// TIA Portal project "TIA portal v16_V16" (V16)
// Vorlageprojekt für das Buch mit Zielsystem S7-1200

(* hardware
DEVICE "S7-1200 station_1"  S7-1200 Station
   slot 0: "Rack_0"  S7-1200 Rack  Rack  V1.0
   slot 1: "PLC_2"  CPU 1215C DC/DC/DC  6ES7 215-1AG40-0XB0  V4.4
   slot 2: "DI 16/DQ 16x24VDC_1"  6ES7 223-1BL32-0XB0  V2.0
   slot 3: "DI 16x24VDC_1"  6ES7 221-1BH32-0XB0  V2.0
   slot 4: "AI 4x13BIT/AQ 2x14BIT_1"  6ES7 234-4HE32-0XB0  V2.1
*)

// ===== PLC "PLC_2"  CPU 1215C DC/DC/DC =====

VAR_GLOBAL   // PLC tag table "Default tag table"
   "Security Relay" AT %I0.0 : Bool;
   "Emergency stop feeding" AT %I0.1 : Bool;
   "Emergency stop elevator" AT %I0.2 : Bool;
   "Emergency stop load beld" AT %I0.3 : Bool;
   "Select auto" AT %I0.4 : Bool;
   "Select manual" AT %I0.5 : Bool;
   "Fault reset button" AT %I0.6 : Bool;
   "Manual box feeding button" AT %I1.0 : Bool;
   "Manual load beld" AT %I1.1 : Bool;
   "Manual Clamp" AT %I1.2 : Bool;
   "Box feeder motor guard" AT %I2.0 : Bool;
   "Enable load beld motor guard" AT %I2.1 : Bool;
   "Elevator motor guard" AT %I2.2 : Bool;
   "Load pallet motor guard" AT %I2.3 : Bool;
   "Pallet feeder motor guard" AT %I2.4 : Bool;
   "Exit conveyor motor guard" AT %I2.5 : Bool;
   "Box feeder motor feedback" AT %I3.0 : Bool;
   "Enable load beld motor feedback" AT %I3.1 : Bool;
   "Elevator motor feedback up" AT %I3.2 : Bool;
   "Elevator motor feedback down" AT %I3.3 : Bool;
   "Load pallet motor feedback" AT %I3.4 : Bool;
   "Pallet feeder motor feedback" AT %I3.5 : Bool;
   "Exit conveyor motor feedback" AT %I3.6 : Bool;
   "Pallet at entry" AT %I4.0 : Bool;
   "Pallet at exit" AT %I4.1 : Bool;
   "Pallet loaded" AT %I4.2 : Bool;
   "Up load pallet" AT %I4.3 : Bool;
   "Down load pallet" AT %I4.4 : Bool;
   "Box at entry" AT %I4.5 : Bool;
   "Pusher limit" AT %I4.6 : Bool;
   "Plate limit" AT %I4.7 : Bool;
   "Clamped" AT %I5.0 : Bool;
   "Relay warning ligth" AT %Q0.0 : Bool;
   "Relay aux turn valve" AT %Q0.1 : Bool;
   "Relay aux push valve" AT %Q0.2 : Bool;
   "Relay aux plate valve" AT %Q0.3 : Bool;
   "Relay Clamp" AT %Q0.4 : Bool;
   "Move to limit" AT %Q0.5 : Bool;
   "Enable pallet emiter" AT %Q0.6 : Bool;
   "Enable exit conveyor" AT %Q0.7 : Bool;
   "Enable box feeder motor" AT %Q2.0 : Bool;
   "Enable load beld motor" AT %Q2.1 : Bool;
   "Enable elevator up motor" AT %Q2.2 : Bool;
   "Enable elevator down motor" AT %Q2.3 : Bool;
   "Enable Load pallet motor" AT %Q2.4 : Bool;
   "Enable Pallet feeder motor" AT %Q2.5 : Bool;
   "Enable exit conveyor motor" AT %Q2.6 : Bool;
   "Fault reset light" AT %Q3.0 : Bool;
   "Start feeding light" AT %Q3.1 : Bool;
   "Stop feeding light" AT %Q3.2 : Bool;
   "Counter box" AT %QW50 : Word;
   "Input_Security_Relay" AT %M0.0 : Bool;
   "Input_Emergency_stop_feeding" AT %M0.1 : Bool;
   "Input_emergency_stop_elevator" AT %M0.2 : Bool;
   "Input_emergency_stop_load_beld" AT %M0.3 : Bool;
   "Input_select_auto" AT %M0.4 : Bool;
   "Input_select_manual" AT %M0.5 : Bool;
   "Input_Fault_reset_button" AT %M0.6 : Bool;
   "Input_manual_box_feeding_button" AT %M1.0 : Bool;
   "Input_manual_load_beld" AT %M1.1 : Bool;
   "Input_manual_clamp" AT %M1.2 : Bool;
   "Input_manual_pallet_feeder" AT %M1.3 : Bool;
   "Input_box_feeder_motor_guard" AT %M2.0 : Bool;
   "Input_enable_load_beld_motor_guard" AT %M2.1 : Bool;
   "Input_elevator_motor_guard" AT %M2.2 : Bool;
   "Input_load_pallet_motor_guard" AT %M2.3 : Bool;
   "Input_pallet_feeder_motor_guad" AT %M2.4 : Bool;
   "Input_box_feeder_motor_feedback" AT %M3.0 : Bool;
   "Input_enable_load_beld_motor_feedback" AT %M3.1 : Bool;
   "Input_elevator_motor_feedback_up" AT %M3.2 : Bool;
   "Input_elevator_motor_feedback_down" AT %M3.3 : Bool;
   "Input_load_pallet_motor_feedback" AT %M3.4 : Bool;
   "Input_pallet_feeder_motor_feedback" AT %M3.5 : Bool;
   "Input_pallet_at_entry" AT %M4.0 : Bool;
   "Input_pallet_at_exit" AT %M4.1 : Bool;
   "Input_pallet_loaded" AT %M4.2 : Bool;
   "Input_up_load_pallet" AT %M4.3 : Bool;
   "Input_down_load_pallet" AT %M4.4 : Bool;
   "Input_box_at_entry" AT %M4.5 : Bool;
   "Input_pusher_limit" AT %M4.6 : Bool;
   "Input_plate_limit" AT %M4.7 : Bool;
   "Input_clamped" AT %M5.0 : Bool;
   "Output_warning_ligth" AT %M10.0 : Bool;
   "Output_relay_aux_turn_valve" AT %M10.1 : Bool;
   "Ouput_relay_aux_push_valve" AT %M10.2 : Bool;
   "Output_relay_aux_plate_valve" AT %M10.3 : Bool;
   "Output_relay_clamp" AT %M10.4 : Bool;
   "Ouput_move_to_limit" AT %M10.5 : Bool;
   "Output_enable_pallet_emiter" AT %M10.6 : Bool;
   "Output_enable_exit_conveyor" AT %M10.7 : Bool;
   "Output_enable_box_feeder_motor" AT %M12.0 : Bool;
   "Output_enable_load_beld_motor" AT %M12.1 : Bool;
   "Output_enable_elevator_up_motor" AT %M12.2 : Bool;
   "Output_enable_elevator_down_motor" AT %M12.3 : Bool;
   "Output_enable_load_pallet_motor" AT %M12.4 : Bool;
   "Output_enable_pallet_feeder_motor" AT %M12.5 : Bool;
   "Output_enable_exit_conveyor_motor" AT %M12.6 : Bool;
   "Output_fault_reset_light" AT %M13.0 : Bool;
   "Output_start_feeding_light" AT %M13.1 : Bool;
   "Output_stop_feeding_light" AT %M13.2 : Bool;
   "Ouput_counter_box" AT %MW100 : Word;
   "Emergency_enable" AT %M30.0 : Bool;
   "Manual_box_feeding_drive" AT %M30.1 : Bool;
   "Manual pallet feeder" AT %I1.3 : Bool;
   "Manual load pallet" AT %I1.4 : Bool;
   "Input_manual_load_pallet" AT %M1.4 : Bool;
   "Input_manual_exit_conveyor" AT %M1.5 : Bool;
   "Manual_load_beld_drive" AT %M30.2 : Bool;
   "Manual_clamp_drive" AT %M30.3 : Bool;
   "Manual_pallet_feeder_drive" AT %M30.4 : Bool;
   "Elevator moving" AT %I5.1 : Bool;
   "Manual exit conveyor" AT %I1.5 : Bool;
   "Manual elevator up" AT %I5.2 : Bool;
   "Manual elevator down" AT %I5.3 : Bool;
   "Input_elevator_moving" AT %M5.1 : Bool;
   "Input_manual_elevator_up" AT %M5.2 : Bool;
   "Input_manual_elevator_down" AT %M5.3 : Bool;
   "Manual_load_pallet_drive" AT %M30.5 : Bool;
   "Manual_exit_conveyor_drive" AT %M30.6 : Bool;
   "Manual_elevator_up_drive" AT %M30.7 : Bool;
   "Manual_elevator_down_drive" AT %M31.0 : Bool;
   "Input_exit_conveyor_motor_guard" AT %M2.5 : Bool;
   "Input_exit_conveyor_motor_feedback" AT %M3.6 : Bool;
   "Aux_manual_box_feeding_drive" AT %M31.1 : Bool;
   "Up_manual_box_feeding_drive" AT %M6.0 : Bool;
   "Up_manual_load_beld_drive" AT %M6.1 : Bool;
   "Aux_manual_load_beld_drive" AT %M31.2 : Bool;
   "Aux_manual_pallet_feeder_drive" AT %M31.4 : Bool;
   "Aux_manual_load_pallet_drive" AT %M31.5 : Bool;
   "Aux_manual_exit_conveyor_drive" AT %M31.6 : Bool;
   "Aux_manual_elevator_up_drive" AT %M31.7 : Bool;
   "Aux_manual_elevator_down_drive" AT %M32.0 : Bool;
   "Up_manual_pallet_feeder_drive" AT %M6.2 : Bool;
   "Up_manual_load_pallet_drive" AT %M6.3 : Bool;
   "Up_manual_exit_conveyor_drive" AT %M6.4 : Bool;
   "Up_manual_elevator_up_drive" AT %M6.5 : Bool;
   "Up_manual_elevator_down_drive" AT %M6.6 : Bool;
END_VAR

DATA_BLOCK "Engine_starter_DB_box_feeder"   // DB1
{ S7_Optimized_Access := 'TRUE' }
VERSION : 0.1
// stored: InstanceOfName Engine_starter
"Engine_starter"
BEGIN
END_DATA_BLOCK

DATA_BLOCK "Engine_starter_DB_load_beld"   // DB2
{ S7_Optimized_Access := 'TRUE' }
VERSION : 0.1
// stored: InstanceOfName Engine_starter
"Engine_starter"
BEGIN
END_DATA_BLOCK

DATA_BLOCK "Engine_starter_DB_elevator_up"   // DB3
{ S7_Optimized_Access := 'TRUE' }
VERSION : 0.1
// stored: InstanceOfName Engine_starter
"Engine_starter"
BEGIN
END_DATA_BLOCK

DATA_BLOCK "Engine_starter_DB_elevator_down"   // DB4
{ S7_Optimized_Access := 'TRUE' }
VERSION : 0.1
// stored: InstanceOfName Engine_starter
"Engine_starter"
BEGIN
END_DATA_BLOCK

DATA_BLOCK "Engine_starter_DB_load_pallet"   // DB5
{ S7_Optimized_Access := 'TRUE' }
VERSION : 0.1
// stored: InstanceOfName Engine_starter
"Engine_starter"
BEGIN
END_DATA_BLOCK

DATA_BLOCK "Engine_starter_DB_pallet_feeder"   // DB6
{ S7_Optimized_Access := 'TRUE' }
VERSION : 0.1
// stored: InstanceOfName Engine_starter
"Engine_starter"
BEGIN
END_DATA_BLOCK

DATA_BLOCK "Engine_starter_DB_exit_conveyor"   // DB7
{ S7_Optimized_Access := 'TRUE' }
VERSION : 0.1
// stored: InstanceOfName Engine_starter
"Engine_starter"
BEGIN
END_DATA_BLOCK

FUNCTION_BLOCK "Engine_starter"   // FB1, LAD
{ S7_Optimized_Access := 'TRUE' }
VERSION : 0.1
   VAR_INPUT
      STOP_EMERGENCY : Bool;
      THERMAL_SHUTDOWN : Bool;
      CONTACT_FEEDBACK : Bool;
      ENABLE : Bool;
      RESET_FAULT : Bool;
   END_VAR
   VAR_OUTPUT
      START_ENABLED : Bool;
      STARTING_FAILURE : Bool;
      ACTIVE_EMERGENCY : Bool;
      ACTIVE_THERMAL : Bool;
      FEEDBACK_FAILURE : Bool;
   END_VAR
   VAR
      stop_error : Bool;
      temp_feedback : TON_TIME;
      enable_engine : Bool;
      temp_thermal_shutdown : TON_TIME;
   END_VAR
BEGIN

REGION Network 1
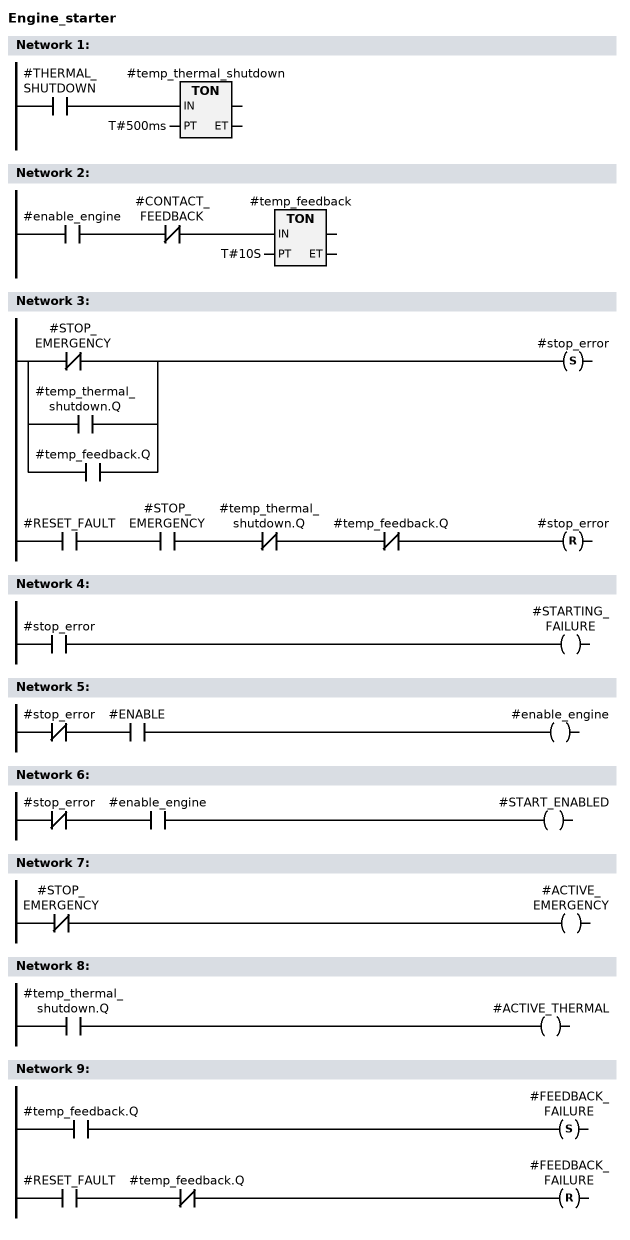
   #temp_thermal_shutdown(IN := #THERMAL_SHUTDOWN, PT := T#500ms);   // TON
END_REGION

REGION Network 2
   #temp_feedback(IN := #enable_engine AND NOT #CONTACT_FEEDBACK, PT := T#10S);   // TON
END_REGION

REGION Network 3
   RUNG wire#powerrail
      I_Contact( #STOP_EMERGENCY )
      wire#w1
      S_Coil( #stop_error )
   END_RUNG
   RUNG wire#powerrail
      Contact( #temp_thermal_shutdown.Q )
   END_RUNG wire#w1
   RUNG wire#powerrail
      Contact( #temp_feedback.Q )
   END_RUNG wire#w1
   RUNG wire#powerrail
      Contact( #RESET_FAULT )
      Contact( #STOP_EMERGENCY )
      I_Contact( #temp_thermal_shutdown.Q )
      I_Contact( #temp_feedback.Q )
      R_Coil( #stop_error )
   END_RUNG
   // the same network as SCL:
   IF NOT #STOP_EMERGENCY OR #temp_thermal_shutdown.Q OR #temp_feedback.Q THEN #stop_error := TRUE; END_IF;
   IF #RESET_FAULT AND #STOP_EMERGENCY AND NOT #temp_thermal_shutdown.Q AND NOT #temp_feedback.Q THEN
       #stop_error := FALSE;
   END_IF;
END_REGION

REGION Network 4
   RUNG wire#powerrail
      Contact( #stop_error )
      Coil( #STARTING_FAILURE )
   END_RUNG
   // the same network as SCL:
   #STARTING_FAILURE := #stop_error;
END_REGION

REGION Network 5
   RUNG wire#powerrail
      I_Contact( #stop_error )
      Contact( #ENABLE )
      Coil( #enable_engine )
   END_RUNG
   // the same network as SCL:
   #enable_engine := NOT #stop_error AND #ENABLE;
END_REGION

REGION Network 6
   RUNG wire#powerrail
      I_Contact( #stop_error )
      Contact( #enable_engine )
      Coil( #START_ENABLED )
   END_RUNG
   // the same network as SCL:
   #START_ENABLED := NOT #stop_error AND #enable_engine;
END_REGION

REGION Network 7
   RUNG wire#powerrail
      I_Contact( #STOP_EMERGENCY )
      Coil( #ACTIVE_EMERGENCY )
   END_RUNG
   // the same network as SCL:
   #ACTIVE_EMERGENCY := NOT #STOP_EMERGENCY;
END_REGION

REGION Network 8
   RUNG wire#powerrail
      Contact( #temp_thermal_shutdown.Q )
      Coil( #ACTIVE_THERMAL )
   END_RUNG
   // the same network as SCL:
   #ACTIVE_THERMAL := #temp_thermal_shutdown.Q;
END_REGION

REGION Network 9
   RUNG wire#powerrail
      Contact( #temp_feedback.Q )
      S_Coil( #FEEDBACK_FAILURE )
   END_RUNG
   RUNG wire#powerrail
      Contact( #RESET_FAULT )
      I_Contact( #temp_feedback.Q )
      R_Coil( #FEEDBACK_FAILURE )
   END_RUNG
   // the same network as SCL:
   IF #temp_feedback.Q THEN #FEEDBACK_FAILURE := TRUE; END_IF;
   IF #RESET_FAULT AND NOT #temp_feedback.Q THEN #FEEDBACK_FAILURE := FALSE; END_IF;
END_REGION
END_FUNCTION_BLOCK

FUNCTION "Input_Management" : Void   // FC1, LAD
{ S7_Optimized_Access := 'TRUE' }
VERSION : 0.1
BEGIN

REGION Network 1
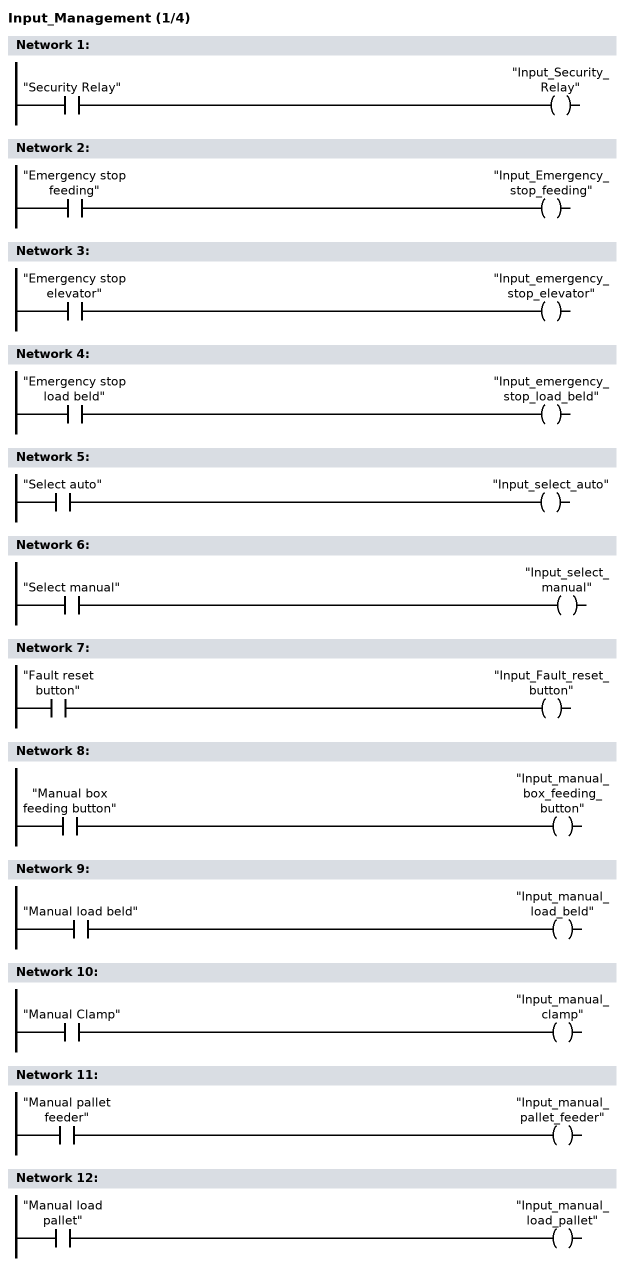
   RUNG wire#powerrail
      Contact( "Security Relay" )
      Coil( "Input_Security_Relay" )
   END_RUNG
   // the same network as SCL:
   "Input_Security_Relay" := "Security Relay";
END_REGION

REGION Network 2
   RUNG wire#powerrail
      Contact( "Emergency stop feeding" )
      Coil( "Input_Emergency_stop_feeding" )
   END_RUNG
   // the same network as SCL:
   "Input_Emergency_stop_feeding" := "Emergency stop feeding";
END_REGION

REGION Network 3
   RUNG wire#powerrail
      Contact( "Emergency stop elevator" )
      Coil( "Input_emergency_stop_elevator" )
   END_RUNG
   // the same network as SCL:
   "Input_emergency_stop_elevator" := "Emergency stop elevator";
END_REGION

REGION Network 4
   RUNG wire#powerrail
      Contact( "Emergency stop load beld" )
      Coil( "Input_emergency_stop_load_beld" )
   END_RUNG
   // the same network as SCL:
   "Input_emergency_stop_load_beld" := "Emergency stop load beld";
END_REGION

REGION Network 5
   RUNG wire#powerrail
      Contact( "Select auto" )
      Coil( "Input_select_auto" )
   END_RUNG
   // the same network as SCL:
   "Input_select_auto" := "Select auto";
END_REGION

REGION Network 6
   RUNG wire#powerrail
      Contact( "Select manual" )
      Coil( "Input_select_manual" )
   END_RUNG
   // the same network as SCL:
   "Input_select_manual" := "Select manual";
END_REGION

REGION Network 7
   RUNG wire#powerrail
      Contact( "Fault reset button" )
      Coil( "Input_Fault_reset_button" )
   END_RUNG
   // the same network as SCL:
   "Input_Fault_reset_button" := "Fault reset button";
END_REGION

REGION Network 8
   RUNG wire#powerrail
      Contact( "Manual box feeding button" )
      Coil( "Input_manual_box_feeding_button" )
   END_RUNG
   // the same network as SCL:
   "Input_manual_box_feeding_button" := "Manual box feeding button";
END_REGION

REGION Network 9
   RUNG wire#powerrail
      Contact( "Manual load beld" )
      Coil( "Input_manual_load_beld" )
   END_RUNG
   // the same network as SCL:
   "Input_manual_load_beld" := "Manual load beld";
END_REGION

REGION Network 10
   RUNG wire#powerrail
      Contact( "Manual Clamp" )
      Coil( "Input_manual_clamp" )
   END_RUNG
   // the same network as SCL:
   "Input_manual_clamp" := "Manual Clamp";
END_REGION

REGION Network 11
   RUNG wire#powerrail
      Contact( "Manual pallet feeder" )
      Coil( "Input_manual_pallet_feeder" )
   END_RUNG
   // the same network as SCL:
   "Input_manual_pallet_feeder" := "Manual pallet feeder";
END_REGION

REGION Network 12
   RUNG wire#powerrail
      Contact( "Manual load pallet" )
      Coil( "Input_manual_load_pallet" )
   END_RUNG
   // the same network as SCL:
   "Input_manual_load_pallet" := "Manual load pallet";
END_REGION

REGION Network 13
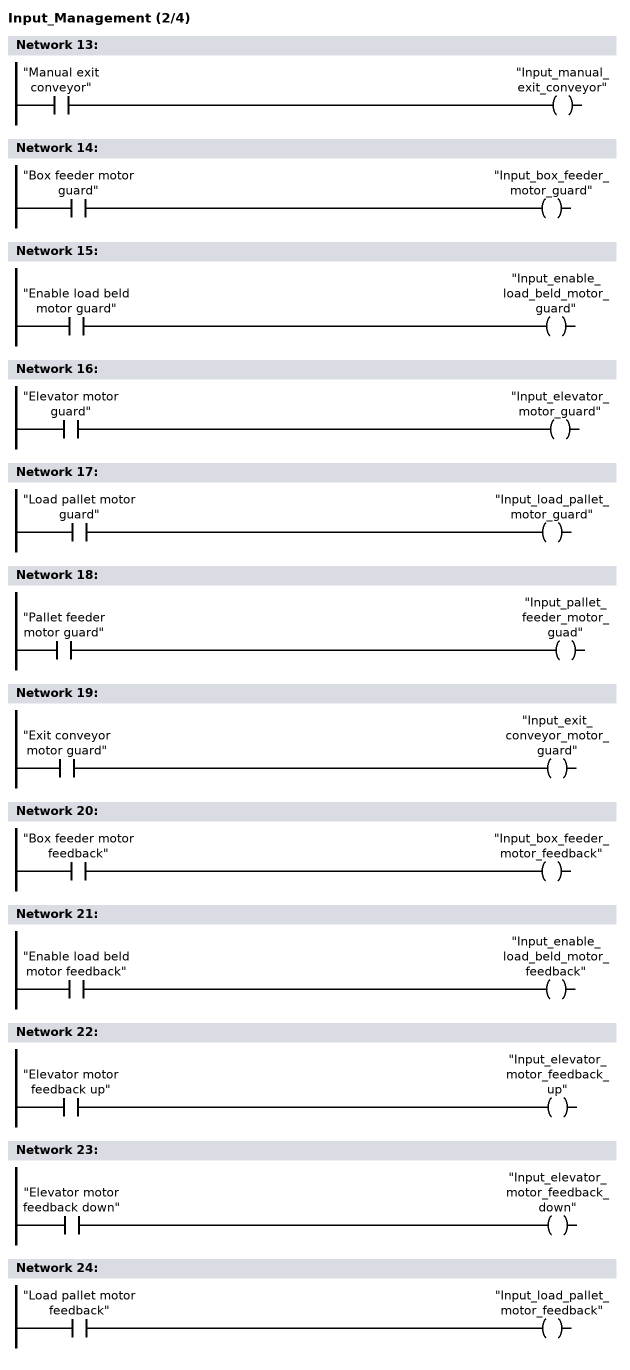
   RUNG wire#powerrail
      Contact( "Manual exit conveyor" )
      Coil( "Input_manual_exit_conveyor" )
   END_RUNG
   // the same network as SCL:
   "Input_manual_exit_conveyor" := "Manual exit conveyor";
END_REGION

REGION Network 14
   RUNG wire#powerrail
      Contact( "Box feeder motor guard" )
      Coil( "Input_box_feeder_motor_guard" )
   END_RUNG
   // the same network as SCL:
   "Input_box_feeder_motor_guard" := "Box feeder motor guard";
END_REGION

REGION Network 15
   RUNG wire#powerrail
      Contact( "Enable load beld motor guard" )
      Coil( "Input_enable_load_beld_motor_guard" )
   END_RUNG
   // the same network as SCL:
   "Input_enable_load_beld_motor_guard" := "Enable load beld motor guard";
END_REGION

REGION Network 16
   RUNG wire#powerrail
      Contact( "Elevator motor guard" )
      Coil( "Input_elevator_motor_guard" )
   END_RUNG
   // the same network as SCL:
   "Input_elevator_motor_guard" := "Elevator motor guard";
END_REGION

REGION Network 17
   RUNG wire#powerrail
      Contact( "Load pallet motor guard" )
      Coil( "Input_load_pallet_motor_guard" )
   END_RUNG
   // the same network as SCL:
   "Input_load_pallet_motor_guard" := "Load pallet motor guard";
END_REGION

REGION Network 18
   RUNG wire#powerrail
      Contact( "Pallet feeder motor guard" )
      Coil( "Input_pallet_feeder_motor_guad" )
   END_RUNG
   // the same network as SCL:
   "Input_pallet_feeder_motor_guad" := "Pallet feeder motor guard";
END_REGION

REGION Network 19
   RUNG wire#powerrail
      Contact( "Exit conveyor motor guard" )
      Coil( "Input_exit_conveyor_motor_guard" )
   END_RUNG
   // the same network as SCL:
   "Input_exit_conveyor_motor_guard" := "Exit conveyor motor guard";
END_REGION

REGION Network 20
   RUNG wire#powerrail
      Contact( "Box feeder motor feedback" )
      Coil( "Input_box_feeder_motor_feedback" )
   END_RUNG
   // the same network as SCL:
   "Input_box_feeder_motor_feedback" := "Box feeder motor feedback";
END_REGION

REGION Network 21
   RUNG wire#powerrail
      Contact( "Enable load beld motor feedback" )
      Coil( "Input_enable_load_beld_motor_feedback" )
   END_RUNG
   // the same network as SCL:
   "Input_enable_load_beld_motor_feedback" := "Enable load beld motor feedback";
END_REGION

REGION Network 22
   RUNG wire#powerrail
      Contact( "Elevator motor feedback up" )
      Coil( "Input_elevator_motor_feedback_up" )
   END_RUNG
   // the same network as SCL:
   "Input_elevator_motor_feedback_up" := "Elevator motor feedback up";
END_REGION

REGION Network 23
   RUNG wire#powerrail
      Contact( "Elevator motor feedback down" )
      Coil( "Input_elevator_motor_feedback_down" )
   END_RUNG
   // the same network as SCL:
   "Input_elevator_motor_feedback_down" := "Elevator motor feedback down";
END_REGION

REGION Network 24
   RUNG wire#powerrail
      Contact( "Load pallet motor feedback" )
      Coil( "Input_load_pallet_motor_feedback" )
   END_RUNG
   // the same network as SCL:
   "Input_load_pallet_motor_feedback" := "Load pallet motor feedback";
END_REGION

REGION Network 25
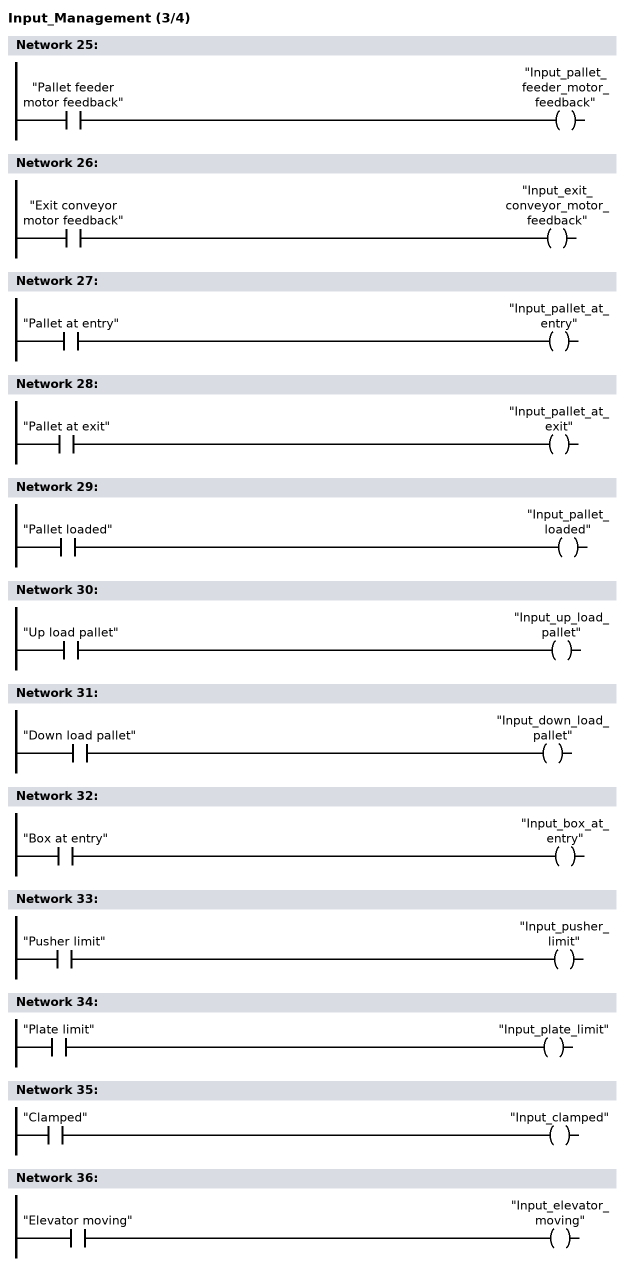
   RUNG wire#powerrail
      Contact( "Pallet feeder motor feedback" )
      Coil( "Input_pallet_feeder_motor_feedback" )
   END_RUNG
   // the same network as SCL:
   "Input_pallet_feeder_motor_feedback" := "Pallet feeder motor feedback";
END_REGION

REGION Network 26
   RUNG wire#powerrail
      Contact( "Exit conveyor motor feedback" )
      Coil( "Input_exit_conveyor_motor_feedback" )
   END_RUNG
   // the same network as SCL:
   "Input_exit_conveyor_motor_feedback" := "Exit conveyor motor feedback";
END_REGION

REGION Network 27
   RUNG wire#powerrail
      Contact( "Pallet at entry" )
      Coil( "Input_pallet_at_entry" )
   END_RUNG
   // the same network as SCL:
   "Input_pallet_at_entry" := "Pallet at entry";
END_REGION

REGION Network 28
   RUNG wire#powerrail
      Contact( "Pallet at exit" )
      Coil( "Input_pallet_at_exit" )
   END_RUNG
   // the same network as SCL:
   "Input_pallet_at_exit" := "Pallet at exit";
END_REGION

REGION Network 29
   RUNG wire#powerrail
      Contact( "Pallet loaded" )
      Coil( "Input_pallet_loaded" )
   END_RUNG
   // the same network as SCL:
   "Input_pallet_loaded" := "Pallet loaded";
END_REGION

REGION Network 30
   RUNG wire#powerrail
      Contact( "Up load pallet" )
      Coil( "Input_up_load_pallet" )
   END_RUNG
   // the same network as SCL:
   "Input_up_load_pallet" := "Up load pallet";
END_REGION

REGION Network 31
   RUNG wire#powerrail
      Contact( "Down load pallet" )
      Coil( "Input_down_load_pallet" )
   END_RUNG
   // the same network as SCL:
   "Input_down_load_pallet" := "Down load pallet";
END_REGION

REGION Network 32
   RUNG wire#powerrail
      Contact( "Box at entry" )
      Coil( "Input_box_at_entry" )
   END_RUNG
   // the same network as SCL:
   "Input_box_at_entry" := "Box at entry";
END_REGION

REGION Network 33
   RUNG wire#powerrail
      Contact( "Pusher limit" )
      Coil( "Input_pusher_limit" )
   END_RUNG
   // the same network as SCL:
   "Input_pusher_limit" := "Pusher limit";
END_REGION

REGION Network 34
   RUNG wire#powerrail
      Contact( "Plate limit" )
      Coil( "Input_plate_limit" )
   END_RUNG
   // the same network as SCL:
   "Input_plate_limit" := "Plate limit";
END_REGION

REGION Network 35
   RUNG wire#powerrail
      Contact( "Clamped" )
      Coil( "Input_clamped" )
   END_RUNG
   // the same network as SCL:
   "Input_clamped" := "Clamped";
END_REGION

REGION Network 36
   RUNG wire#powerrail
      Contact( "Elevator moving" )
      Coil( "Input_elevator_moving" )
   END_RUNG
   // the same network as SCL:
   "Input_elevator_moving" := "Elevator moving";
END_REGION

REGION Network 37
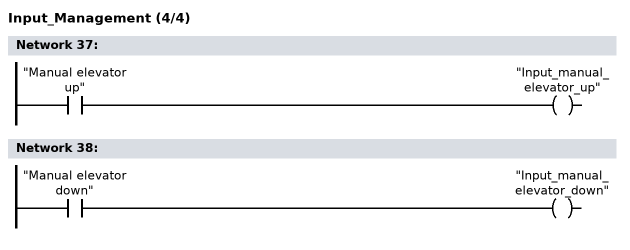
   RUNG wire#powerrail
      Contact( "Manual elevator up" )
      Coil( "Input_manual_elevator_up" )
   END_RUNG
   // the same network as SCL:
   "Input_manual_elevator_up" := "Manual elevator up";
END_REGION

REGION Network 38
   RUNG wire#powerrail
      Contact( "Manual elevator down" )
      Coil( "Input_manual_elevator_down" )
   END_RUNG
   // the same network as SCL:
   "Input_manual_elevator_down" := "Manual elevator down";
END_REGION
END_FUNCTION

FUNCTION "Output_Management" : Void   // FC2, LAD
{ S7_Optimized_Access := 'TRUE' }
VERSION : 0.1
BEGIN

REGION Network 1
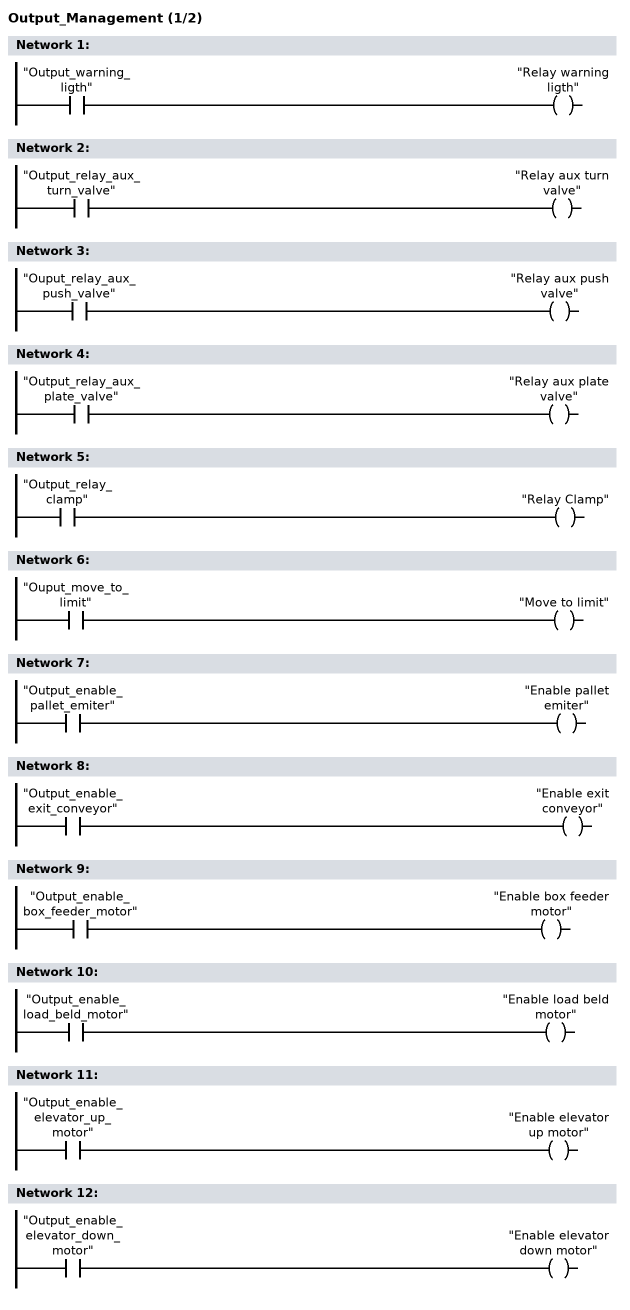
   RUNG wire#powerrail
      Contact( "Output_warning_ligth" )
      Coil( "Relay warning ligth" )
   END_RUNG
   // the same network as SCL:
   "Relay warning ligth" := "Output_warning_ligth";
END_REGION

REGION Network 2
   RUNG wire#powerrail
      Contact( "Output_relay_aux_turn_valve" )
      Coil( "Relay aux turn valve" )
   END_RUNG
   // the same network as SCL:
   "Relay aux turn valve" := "Output_relay_aux_turn_valve";
END_REGION

REGION Network 3
   RUNG wire#powerrail
      Contact( "Ouput_relay_aux_push_valve" )
      Coil( "Relay aux push valve" )
   END_RUNG
   // the same network as SCL:
   "Relay aux push valve" := "Ouput_relay_aux_push_valve";
END_REGION

REGION Network 4
   RUNG wire#powerrail
      Contact( "Output_relay_aux_plate_valve" )
      Coil( "Relay aux plate valve" )
   END_RUNG
   // the same network as SCL:
   "Relay aux plate valve" := "Output_relay_aux_plate_valve";
END_REGION

REGION Network 5
   RUNG wire#powerrail
      Contact( "Output_relay_clamp" )
      Coil( "Relay Clamp" )
   END_RUNG
   // the same network as SCL:
   "Relay Clamp" := "Output_relay_clamp";
END_REGION

REGION Network 6
   RUNG wire#powerrail
      Contact( "Ouput_move_to_limit" )
      Coil( "Move to limit" )
   END_RUNG
   // the same network as SCL:
   "Move to limit" := "Ouput_move_to_limit";
END_REGION

REGION Network 7
   RUNG wire#powerrail
      Contact( "Output_enable_pallet_emiter" )
      Coil( "Enable pallet emiter" )
   END_RUNG
   // the same network as SCL:
   "Enable pallet emiter" := "Output_enable_pallet_emiter";
END_REGION

REGION Network 8
   RUNG wire#powerrail
      Contact( "Output_enable_exit_conveyor" )
      Coil( "Enable exit conveyor" )
   END_RUNG
   // the same network as SCL:
   "Enable exit conveyor" := "Output_enable_exit_conveyor";
END_REGION

REGION Network 9
   RUNG wire#powerrail
      Contact( "Output_enable_box_feeder_motor" )
      Coil( "Enable box feeder motor" )
   END_RUNG
   // the same network as SCL:
   "Enable box feeder motor" := "Output_enable_box_feeder_motor";
END_REGION

REGION Network 10
   RUNG wire#powerrail
      Contact( "Output_enable_load_beld_motor" )
      Coil( "Enable load beld motor" )
   END_RUNG
   // the same network as SCL:
   "Enable load beld motor" := "Output_enable_load_beld_motor";
END_REGION

REGION Network 11
   RUNG wire#powerrail
      Contact( "Output_enable_elevator_up_motor" )
      Coil( "Enable elevator up motor" )
   END_RUNG
   // the same network as SCL:
   "Enable elevator up motor" := "Output_enable_elevator_up_motor";
END_REGION

REGION Network 12
   RUNG wire#powerrail
      Contact( "Output_enable_elevator_down_motor" )
      Coil( "Enable elevator down motor" )
   END_RUNG
   // the same network as SCL:
   "Enable elevator down motor" := "Output_enable_elevator_down_motor";
END_REGION

REGION Network 13
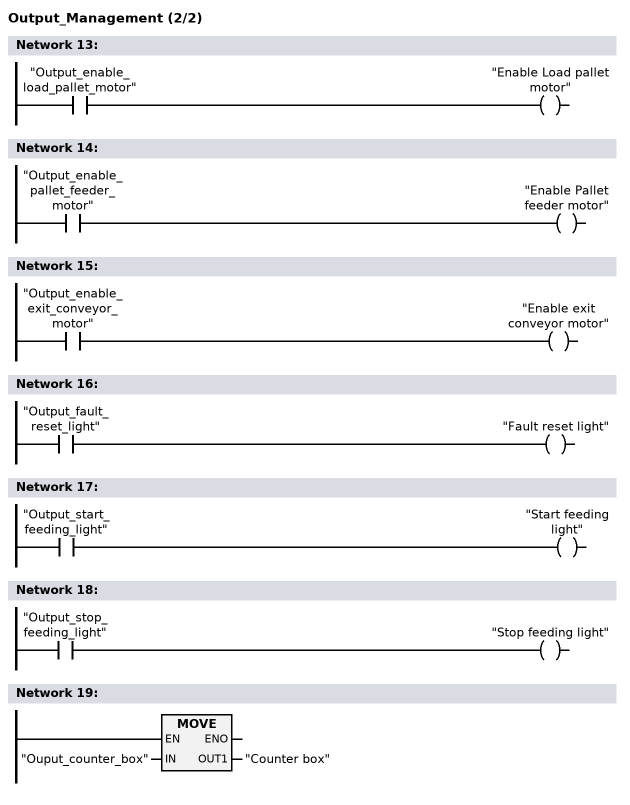
   RUNG wire#powerrail
      Contact( "Output_enable_load_pallet_motor" )
      Coil( "Enable Load pallet motor" )
   END_RUNG
   // the same network as SCL:
   "Enable Load pallet motor" := "Output_enable_load_pallet_motor";
END_REGION

REGION Network 14
   RUNG wire#powerrail
      Contact( "Output_enable_pallet_feeder_motor" )
      Coil( "Enable Pallet feeder motor" )
   END_RUNG
   // the same network as SCL:
   "Enable Pallet feeder motor" := "Output_enable_pallet_feeder_motor";
END_REGION

REGION Network 15
   RUNG wire#powerrail
      Contact( "Output_enable_exit_conveyor_motor" )
      Coil( "Enable exit conveyor motor" )
   END_RUNG
   // the same network as SCL:
   "Enable exit conveyor motor" := "Output_enable_exit_conveyor_motor";
END_REGION

REGION Network 16
   RUNG wire#powerrail
      Contact( "Output_fault_reset_light" )
      Coil( "Fault reset light" )
   END_RUNG
   // the same network as SCL:
   "Fault reset light" := "Output_fault_reset_light";
END_REGION

REGION Network 17
   RUNG wire#powerrail
      Contact( "Output_start_feeding_light" )
      Coil( "Start feeding light" )
   END_RUNG
   // the same network as SCL:
   "Start feeding light" := "Output_start_feeding_light";
END_REGION

REGION Network 18
   RUNG wire#powerrail
      Contact( "Output_stop_feeding_light" )
      Coil( "Stop feeding light" )
   END_RUNG
   // the same network as SCL:
   "Stop feeding light" := "Output_stop_feeding_light";
END_REGION

REGION Network 19
   RUNG wire#powerrail
      Move(in := "Ouput_counter_box", out1 => "Counter box")
   END_RUNG
   // the same network as SCL:
   "Counter box" := "Ouput_counter_box";
END_REGION
END_FUNCTION

FUNCTION "Module_security" : Void   // FC3, LAD
{ S7_Optimized_Access := 'TRUE' }
VERSION : 0.1
BEGIN

REGION Network 1
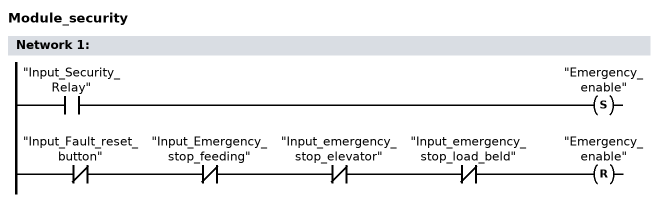
   RUNG wire#powerrail
      Contact( "Input_Security_Relay" )
      S_Coil( "Emergency_enable" )
   END_RUNG
   RUNG wire#powerrail
      I_Contact( "Input_Fault_reset_button" )
      I_Contact( "Input_Emergency_stop_feeding" )
      I_Contact( "Input_emergency_stop_elevator" )
      I_Contact( "Input_emergency_stop_load_beld" )
      R_Coil( "Emergency_enable" )
   END_RUNG
   // the same network as SCL:
   IF "Input_Security_Relay" THEN "Emergency_enable" := TRUE; END_IF;
   IF NOT "Input_Fault_reset_button" AND NOT "Input_Emergency_stop_feeding" AND NOT "Input_emergency_stop_elevator" AND NOT "Input_emergency_stop_load_beld" THEN
       "Emergency_enable" := FALSE;
   END_IF;
END_REGION
END_FUNCTION

FUNCTION "Manual_drive_module" : Void   // FC4, LAD
{ S7_Optimized_Access := 'TRUE' }
VERSION : 0.1
   VAR_TEMP   // added for the SCL form of the ladder/FBD networks
      _w1 : Bool;
   END_VAR
BEGIN

REGION Network 1
   // Manual box feeder
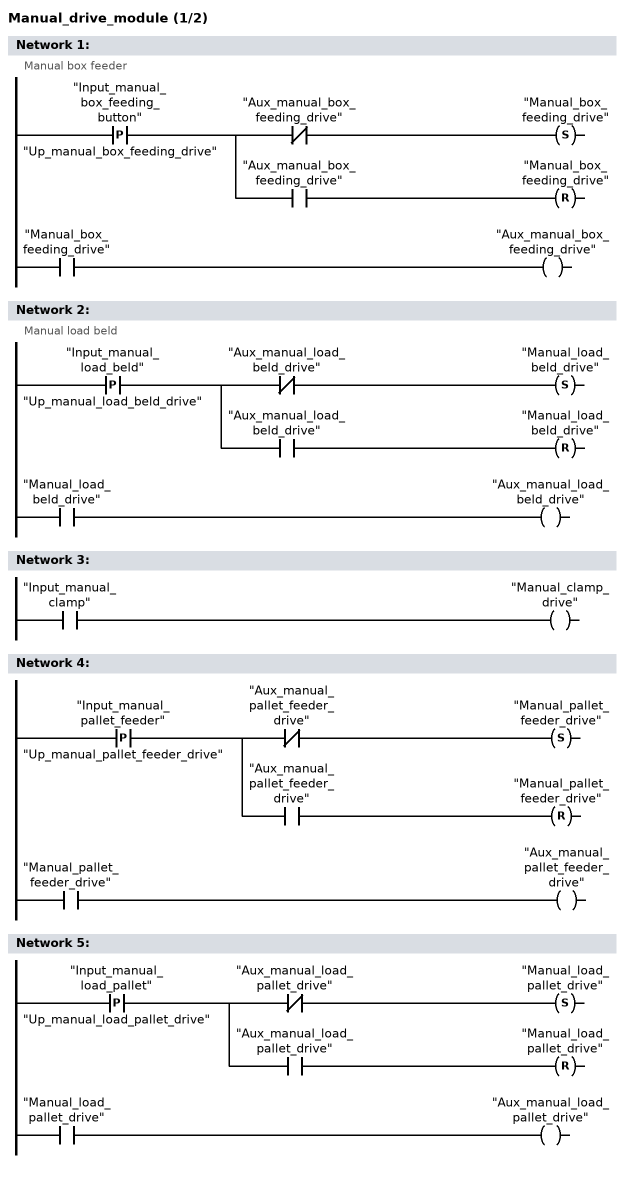
   RUNG wire#powerrail
      P_Contact(operand := "Input_manual_box_feeding_button", bit := "Up_manual_box_feeding_drive")
      wire#w1
      I_Contact( "Aux_manual_box_feeding_drive" )
      S_Coil( "Manual_box_feeding_drive" )
   END_RUNG
   RUNG wire#w1
      Contact( "Aux_manual_box_feeding_drive" )
      R_Coil( "Manual_box_feeding_drive" )
   END_RUNG
   RUNG wire#powerrail
      Contact( "Manual_box_feeding_drive" )
      Coil( "Aux_manual_box_feeding_drive" )
   END_RUNG
   // the same network as SCL:
   #_w1 := "Input_manual_box_feeding_button" AND NOT "Up_manual_box_feeding_drive";   // rising edge of "Input_manual_box_feeding_button"
   "Up_manual_box_feeding_drive" := "Input_manual_box_feeding_button";
   IF #_w1 AND NOT "Aux_manual_box_feeding_drive" THEN "Manual_box_feeding_drive" := TRUE; END_IF;
   IF #_w1 AND "Aux_manual_box_feeding_drive" THEN "Manual_box_feeding_drive" := FALSE; END_IF;
   "Aux_manual_box_feeding_drive" := "Manual_box_feeding_drive";
END_REGION

REGION Network 2
   // Manual load beld
   RUNG wire#powerrail
      P_Contact(operand := "Input_manual_load_beld", bit := "Up_manual_load_beld_drive")
      wire#w1
      I_Contact( "Aux_manual_load_beld_drive" )
      S_Coil( "Manual_load_beld_drive" )
   END_RUNG
   RUNG wire#w1
      Contact( "Aux_manual_load_beld_drive" )
      R_Coil( "Manual_load_beld_drive" )
   END_RUNG
   RUNG wire#powerrail
      Contact( "Manual_load_beld_drive" )
      Coil( "Aux_manual_load_beld_drive" )
   END_RUNG
   // the same network as SCL:
   #_w1 := "Input_manual_load_beld" AND NOT "Up_manual_load_beld_drive";   // rising edge of "Input_manual_load_beld"
   "Up_manual_load_beld_drive" := "Input_manual_load_beld";
   IF #_w1 AND NOT "Aux_manual_load_beld_drive" THEN "Manual_load_beld_drive" := TRUE; END_IF;
   IF #_w1 AND "Aux_manual_load_beld_drive" THEN "Manual_load_beld_drive" := FALSE; END_IF;
   "Aux_manual_load_beld_drive" := "Manual_load_beld_drive";
END_REGION

REGION Network 3
   RUNG wire#powerrail
      Contact( "Input_manual_clamp" )
      Coil( "Manual_clamp_drive" )
   END_RUNG
   // the same network as SCL:
   "Manual_clamp_drive" := "Input_manual_clamp";
END_REGION

REGION Network 4
   RUNG wire#powerrail
      P_Contact(operand := "Input_manual_pallet_feeder", bit := "Up_manual_pallet_feeder_drive")
      wire#w1
      I_Contact( "Aux_manual_pallet_feeder_drive" )
      S_Coil( "Manual_pallet_feeder_drive" )
   END_RUNG
   RUNG wire#w1
      Contact( "Aux_manual_pallet_feeder_drive" )
      R_Coil( "Manual_pallet_feeder_drive" )
   END_RUNG
   RUNG wire#powerrail
      Contact( "Manual_pallet_feeder_drive" )
      Coil( "Aux_manual_pallet_feeder_drive" )
   END_RUNG
   // the same network as SCL:
   #_w1 := "Input_manual_pallet_feeder" AND NOT "Up_manual_pallet_feeder_drive";   // rising edge of "Input_manual_pallet_feeder"
   "Up_manual_pallet_feeder_drive" := "Input_manual_pallet_feeder";
   IF #_w1 AND NOT "Aux_manual_pallet_feeder_drive" THEN "Manual_pallet_feeder_drive" := TRUE; END_IF;
   IF #_w1 AND "Aux_manual_pallet_feeder_drive" THEN "Manual_pallet_feeder_drive" := FALSE; END_IF;
   "Aux_manual_pallet_feeder_drive" := "Manual_pallet_feeder_drive";
END_REGION

REGION Network 5
   RUNG wire#powerrail
      P_Contact(operand := "Input_manual_load_pallet", bit := "Up_manual_load_pallet_drive")
      wire#w1
      I_Contact( "Aux_manual_load_pallet_drive" )
      S_Coil( "Manual_load_pallet_drive" )
   END_RUNG
   RUNG wire#w1
      Contact( "Aux_manual_load_pallet_drive" )
      R_Coil( "Manual_load_pallet_drive" )
   END_RUNG
   RUNG wire#powerrail
      Contact( "Manual_load_pallet_drive" )
      Coil( "Aux_manual_load_pallet_drive" )
   END_RUNG
   // the same network as SCL:
   #_w1 := "Input_manual_load_pallet" AND NOT "Up_manual_load_pallet_drive";   // rising edge of "Input_manual_load_pallet"
   "Up_manual_load_pallet_drive" := "Input_manual_load_pallet";
   IF #_w1 AND NOT "Aux_manual_load_pallet_drive" THEN "Manual_load_pallet_drive" := TRUE; END_IF;
   IF #_w1 AND "Aux_manual_load_pallet_drive" THEN "Manual_load_pallet_drive" := FALSE; END_IF;
   "Aux_manual_load_pallet_drive" := "Manual_load_pallet_drive";
END_REGION

REGION Network 6
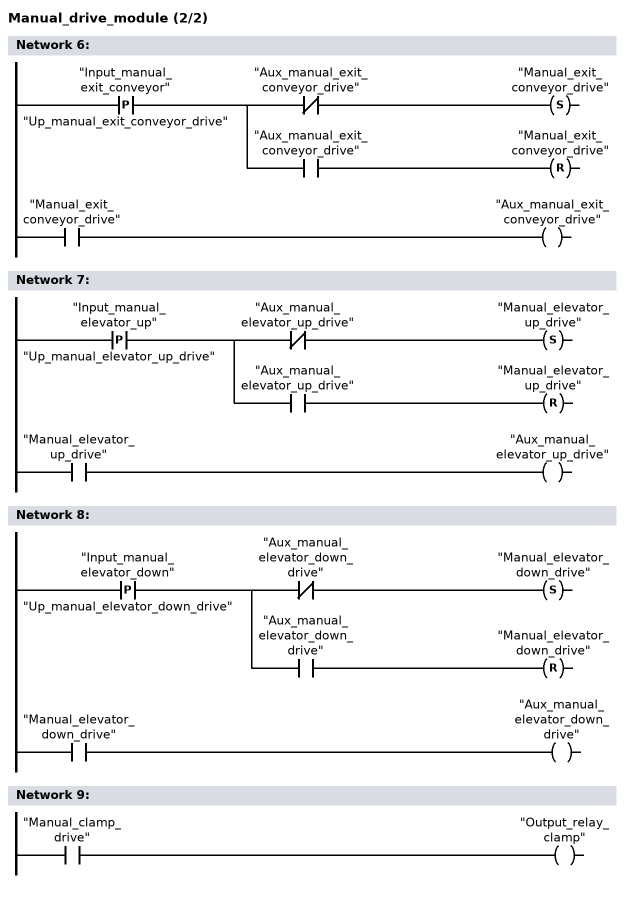
   RUNG wire#powerrail
      P_Contact(operand := "Input_manual_exit_conveyor", bit := "Up_manual_exit_conveyor_drive")
      wire#w1
      I_Contact( "Aux_manual_exit_conveyor_drive" )
      S_Coil( "Manual_exit_conveyor_drive" )
   END_RUNG
   RUNG wire#w1
      Contact( "Aux_manual_exit_conveyor_drive" )
      R_Coil( "Manual_exit_conveyor_drive" )
   END_RUNG
   RUNG wire#powerrail
      Contact( "Manual_exit_conveyor_drive" )
      Coil( "Aux_manual_exit_conveyor_drive" )
   END_RUNG
   // the same network as SCL:
   #_w1 := "Input_manual_exit_conveyor" AND NOT "Up_manual_exit_conveyor_drive";   // rising edge of "Input_manual_exit_conveyor"
   "Up_manual_exit_conveyor_drive" := "Input_manual_exit_conveyor";
   IF #_w1 AND NOT "Aux_manual_exit_conveyor_drive" THEN "Manual_exit_conveyor_drive" := TRUE; END_IF;
   IF #_w1 AND "Aux_manual_exit_conveyor_drive" THEN "Manual_exit_conveyor_drive" := FALSE; END_IF;
   "Aux_manual_exit_conveyor_drive" := "Manual_exit_conveyor_drive";
END_REGION

REGION Network 7
   RUNG wire#powerrail
      P_Contact(operand := "Input_manual_elevator_up", bit := "Up_manual_elevator_up_drive")
      wire#w1
      I_Contact( "Aux_manual_elevator_up_drive" )
      S_Coil( "Manual_elevator_up_drive" )
   END_RUNG
   RUNG wire#w1
      Contact( "Aux_manual_elevator_up_drive" )
      R_Coil( "Manual_elevator_up_drive" )
   END_RUNG
   RUNG wire#powerrail
      Contact( "Manual_elevator_up_drive" )
      Coil( "Aux_manual_elevator_up_drive" )
   END_RUNG
   // the same network as SCL:
   #_w1 := "Input_manual_elevator_up" AND NOT "Up_manual_elevator_up_drive";   // rising edge of "Input_manual_elevator_up"
   "Up_manual_elevator_up_drive" := "Input_manual_elevator_up";
   IF #_w1 AND NOT "Aux_manual_elevator_up_drive" THEN "Manual_elevator_up_drive" := TRUE; END_IF;
   IF #_w1 AND "Aux_manual_elevator_up_drive" THEN "Manual_elevator_up_drive" := FALSE; END_IF;
   "Aux_manual_elevator_up_drive" := "Manual_elevator_up_drive";
END_REGION

REGION Network 8
   RUNG wire#powerrail
      P_Contact(operand := "Input_manual_elevator_down", bit := "Up_manual_elevator_down_drive")
      wire#w1
      I_Contact( "Aux_manual_elevator_down_drive" )
      S_Coil( "Manual_elevator_down_drive" )
   END_RUNG
   RUNG wire#w1
      Contact( "Aux_manual_elevator_down_drive" )
      R_Coil( "Manual_elevator_down_drive" )
   END_RUNG
   RUNG wire#powerrail
      Contact( "Manual_elevator_down_drive" )
      Coil( "Aux_manual_elevator_down_drive" )
   END_RUNG
   // the same network as SCL:
   #_w1 := "Input_manual_elevator_down" AND NOT "Up_manual_elevator_down_drive";   // rising edge of "Input_manual_elevator_down"
   "Up_manual_elevator_down_drive" := "Input_manual_elevator_down";
   IF #_w1 AND NOT "Aux_manual_elevator_down_drive" THEN "Manual_elevator_down_drive" := TRUE; END_IF;
   IF #_w1 AND "Aux_manual_elevator_down_drive" THEN "Manual_elevator_down_drive" := FALSE; END_IF;
   "Aux_manual_elevator_down_drive" := "Manual_elevator_down_drive";
END_REGION

REGION Network 9
   RUNG wire#powerrail
      Contact( "Manual_clamp_drive" )
      Coil( "Output_relay_clamp" )
   END_RUNG
   // the same network as SCL:
   "Output_relay_clamp" := "Manual_clamp_drive";
END_REGION
END_FUNCTION

FUNCTION "Output_drives" : Void   // FC5, LAD
{ S7_Optimized_Access := 'TRUE' }
VERSION : 0.1
BEGIN

REGION Network 1
   // Drive box feeding
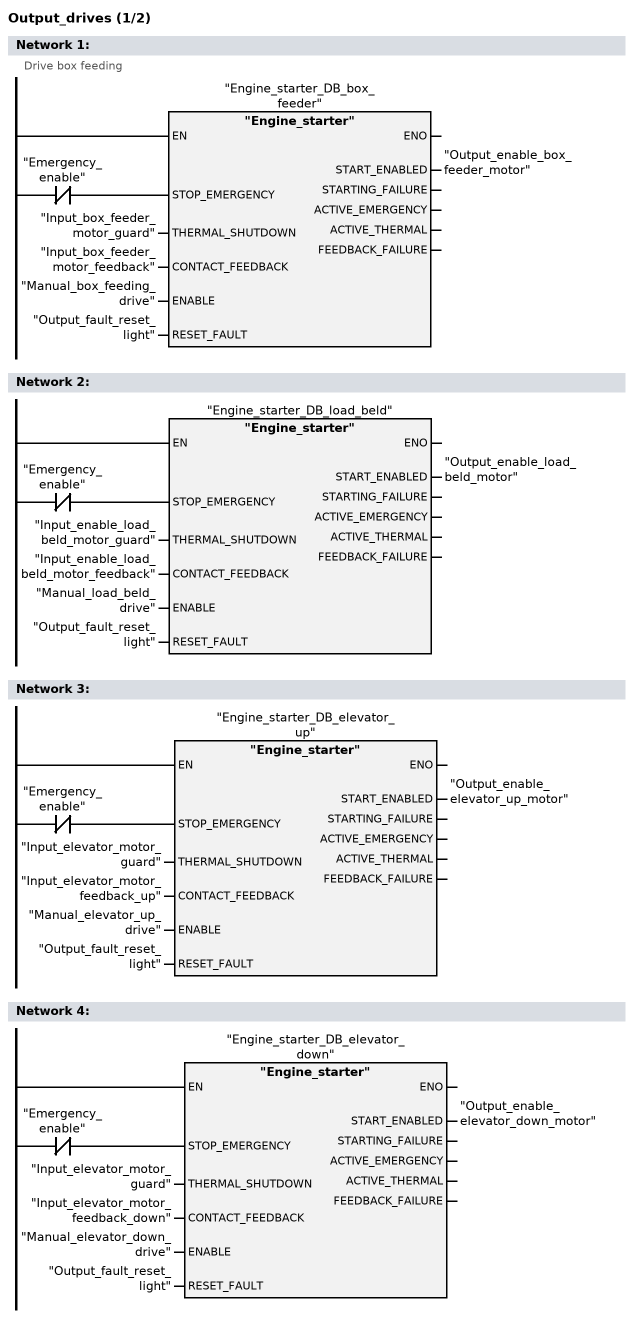
   RUNG wire#powerrail
      "Engine_starter_DB_box_feeder"(STOP_EMERGENCY := wire#w1, THERMAL_SHUTDOWN := "Input_box_feeder_motor_guard", CONTACT_FEEDBACK := "Input_box_feeder_motor_feedback", ENABLE := "Manual_box_feeding_drive", RESET_FAULT := "Output_fault_reset_light", START_ENABLED => "Output_enable_box_feeder_motor", STARTING_FAILURE =>, ACTIVE_EMERGENCY =>, ACTIVE_THERMAL =>, FEEDBACK_FAILURE =>)
   END_RUNG
   RUNG wire#powerrail
      I_Contact( "Emergency_enable" )
   END_RUNG wire#w1
   // the same network as SCL:
   "Engine_starter_DB_box_feeder"(STOP_EMERGENCY := NOT "Emergency_enable",   // "Engine_starter"
                           THERMAL_SHUTDOWN := "Input_box_feeder_motor_guard",
                           CONTACT_FEEDBACK := "Input_box_feeder_motor_feedback",
                           ENABLE := "Manual_box_feeding_drive",
                           RESET_FAULT := "Output_fault_reset_light",
                           START_ENABLED => "Output_enable_box_feeder_motor");
END_REGION

REGION Network 2
   RUNG wire#powerrail
      "Engine_starter_DB_load_beld"(STOP_EMERGENCY := wire#w1, THERMAL_SHUTDOWN := "Input_enable_load_beld_motor_guard", CONTACT_FEEDBACK := "Input_enable_load_beld_motor_feedback", ENABLE := "Manual_load_beld_drive", RESET_FAULT := "Output_fault_reset_light", START_ENABLED => "Output_enable_load_beld_motor", STARTING_FAILURE =>, ACTIVE_EMERGENCY =>, ACTIVE_THERMAL =>, FEEDBACK_FAILURE =>)
   END_RUNG
   RUNG wire#powerrail
      I_Contact( "Emergency_enable" )
   END_RUNG wire#w1
   // the same network as SCL:
   "Engine_starter_DB_load_beld"(STOP_EMERGENCY := NOT "Emergency_enable",   // "Engine_starter"
                           THERMAL_SHUTDOWN := "Input_enable_load_beld_motor_guard",
                           CONTACT_FEEDBACK := "Input_enable_load_beld_motor_feedback",
                           ENABLE := "Manual_load_beld_drive",
                           RESET_FAULT := "Output_fault_reset_light",
                           START_ENABLED => "Output_enable_load_beld_motor");
END_REGION

REGION Network 3
   RUNG wire#powerrail
      "Engine_starter_DB_elevator_up"(STOP_EMERGENCY := wire#w1, THERMAL_SHUTDOWN := "Input_elevator_motor_guard", CONTACT_FEEDBACK := "Input_elevator_motor_feedback_up", ENABLE := "Manual_elevator_up_drive", RESET_FAULT := "Output_fault_reset_light", START_ENABLED => "Output_enable_elevator_up_motor", STARTING_FAILURE =>, ACTIVE_EMERGENCY =>, ACTIVE_THERMAL =>, FEEDBACK_FAILURE =>)
   END_RUNG
   RUNG wire#powerrail
      I_Contact( "Emergency_enable" )
   END_RUNG wire#w1
   // the same network as SCL:
   "Engine_starter_DB_elevator_up"(STOP_EMERGENCY := NOT "Emergency_enable",   // "Engine_starter"
                           THERMAL_SHUTDOWN := "Input_elevator_motor_guard",
                           CONTACT_FEEDBACK := "Input_elevator_motor_feedback_up",
                           ENABLE := "Manual_elevator_up_drive",
                           RESET_FAULT := "Output_fault_reset_light",
                           START_ENABLED => "Output_enable_elevator_up_motor");
END_REGION

REGION Network 4
   RUNG wire#powerrail
      "Engine_starter_DB_elevator_down"(STOP_EMERGENCY := wire#w1, THERMAL_SHUTDOWN := "Input_elevator_motor_guard", CONTACT_FEEDBACK := "Input_elevator_motor_feedback_down", ENABLE := "Manual_elevator_down_drive", RESET_FAULT := "Output_fault_reset_light", START_ENABLED => "Output_enable_elevator_down_motor", STARTING_FAILURE =>, ACTIVE_EMERGENCY =>, ACTIVE_THERMAL =>, FEEDBACK_FAILURE =>)
   END_RUNG
   RUNG wire#powerrail
      I_Contact( "Emergency_enable" )
   END_RUNG wire#w1
   // the same network as SCL:
   "Engine_starter_DB_elevator_down"(STOP_EMERGENCY := NOT "Emergency_enable",   // "Engine_starter"
                           THERMAL_SHUTDOWN := "Input_elevator_motor_guard",
                           CONTACT_FEEDBACK := "Input_elevator_motor_feedback_down",
                           ENABLE := "Manual_elevator_down_drive",
                           RESET_FAULT := "Output_fault_reset_light",
                           START_ENABLED => "Output_enable_elevator_down_motor");
END_REGION

REGION Network 5
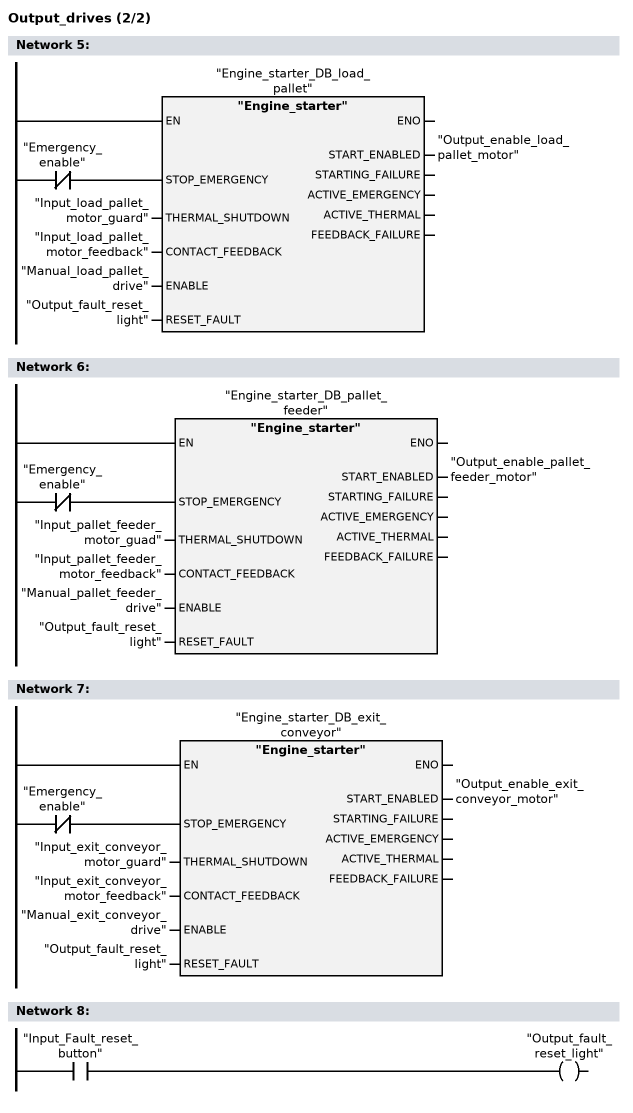
   RUNG wire#powerrail
      "Engine_starter_DB_load_pallet"(STOP_EMERGENCY := wire#w1, THERMAL_SHUTDOWN := "Input_load_pallet_motor_guard", CONTACT_FEEDBACK := "Input_load_pallet_motor_feedback", ENABLE := "Manual_load_pallet_drive", RESET_FAULT := "Output_fault_reset_light", START_ENABLED => "Output_enable_load_pallet_motor", STARTING_FAILURE =>, ACTIVE_EMERGENCY =>, ACTIVE_THERMAL =>, FEEDBACK_FAILURE =>)
   END_RUNG
   RUNG wire#powerrail
      I_Contact( "Emergency_enable" )
   END_RUNG wire#w1
   // the same network as SCL:
   "Engine_starter_DB_load_pallet"(STOP_EMERGENCY := NOT "Emergency_enable",   // "Engine_starter"
                           THERMAL_SHUTDOWN := "Input_load_pallet_motor_guard",
                           CONTACT_FEEDBACK := "Input_load_pallet_motor_feedback",
                           ENABLE := "Manual_load_pallet_drive",
                           RESET_FAULT := "Output_fault_reset_light",
                           START_ENABLED => "Output_enable_load_pallet_motor");
END_REGION

REGION Network 6
   RUNG wire#powerrail
      "Engine_starter_DB_pallet_feeder"(STOP_EMERGENCY := wire#w1, THERMAL_SHUTDOWN := "Input_pallet_feeder_motor_guad", CONTACT_FEEDBACK := "Input_pallet_feeder_motor_feedback", ENABLE := "Manual_pallet_feeder_drive", RESET_FAULT := "Output_fault_reset_light", START_ENABLED => "Output_enable_pallet_feeder_motor", STARTING_FAILURE =>, ACTIVE_EMERGENCY =>, ACTIVE_THERMAL =>, FEEDBACK_FAILURE =>)
   END_RUNG
   RUNG wire#powerrail
      I_Contact( "Emergency_enable" )
   END_RUNG wire#w1
   // the same network as SCL:
   "Engine_starter_DB_pallet_feeder"(STOP_EMERGENCY := NOT "Emergency_enable",   // "Engine_starter"
                           THERMAL_SHUTDOWN := "Input_pallet_feeder_motor_guad",
                           CONTACT_FEEDBACK := "Input_pallet_feeder_motor_feedback",
                           ENABLE := "Manual_pallet_feeder_drive",
                           RESET_FAULT := "Output_fault_reset_light",
                           START_ENABLED => "Output_enable_pallet_feeder_motor");
END_REGION

REGION Network 7
   RUNG wire#powerrail
      "Engine_starter_DB_exit_conveyor"(STOP_EMERGENCY := wire#w1, THERMAL_SHUTDOWN := "Input_exit_conveyor_motor_guard", CONTACT_FEEDBACK := "Input_exit_conveyor_motor_feedback", ENABLE := "Manual_exit_conveyor_drive", RESET_FAULT := "Output_fault_reset_light", START_ENABLED => "Output_enable_exit_conveyor_motor", STARTING_FAILURE =>, ACTIVE_EMERGENCY =>, ACTIVE_THERMAL =>, FEEDBACK_FAILURE =>)
   END_RUNG
   RUNG wire#powerrail
      I_Contact( "Emergency_enable" )
   END_RUNG wire#w1
   // the same network as SCL:
   "Engine_starter_DB_exit_conveyor"(STOP_EMERGENCY := NOT "Emergency_enable",   // "Engine_starter"
                           THERMAL_SHUTDOWN := "Input_exit_conveyor_motor_guard",
                           CONTACT_FEEDBACK := "Input_exit_conveyor_motor_feedback",
                           ENABLE := "Manual_exit_conveyor_drive",
                           RESET_FAULT := "Output_fault_reset_light",
                           START_ENABLED => "Output_enable_exit_conveyor_motor");
END_REGION

REGION Network 8
   RUNG wire#powerrail
      Contact( "Input_Fault_reset_button" )
      Coil( "Output_fault_reset_light" )
   END_RUNG
   // the same network as SCL:
   "Output_fault_reset_light" := "Input_Fault_reset_button";
END_REGION
END_FUNCTION

FUNCTION "MHJ-PLC-Lab-Function-S71200" : Void   // FC9000, SCL
{ S7_Optimized_Access := 'TRUE' }
VERSION : 0.1
   VAR_TEMP
      rdTimeReturn : Int;
      outputTime : DTL;
      SyncVal : Byte;
      forVal : Int;
      forVal_2 : Int;
      Value : Byte;
   END_VAR
   VAR CONSTANT
      CompVal : Byte := 16#34;
      Value_01 : Byte := 16#11;
      Value_01_DW : DWord := 16#A165_D992;
      Value_02_DW : DWord := 16#58BE_4401;
   END_VAR
BEGIN

   #Value:=PEEK(area := 16#82,
        dbNumber := 0,
        byteOffset := 511);
   #Value := #Value + 1;

   POKE(area := 16#82,
        dbNumber := 0,
        byteOffset := 511,
        value := #Value);

   POKE(area:=16#81,
        dbNumber:=0,
        byteOffset:=1016,
        value:=#Value_01_DW);
   POKE(area := 16#81,
        dbNumber := 0,
        byteOffset := 1020,
        value := #Value_02_DW);

   POKE(area := 16#81,
        dbNumber := 0,
        byteOffset := 511,
        value := B#16#00);

   FOR #forVal := 0 TO 120 DO
       FOR #forVal_2:=0 TO 10 DO
           #rdTimeReturn:=RD_SYS_T(#outputTime);
           #rdTimeReturn := WR_SYS_T(#outputTime);
           #rdTimeReturn := RD_SYS_T(#outputTime);
           #rdTimeReturn := WR_SYS_T(#outputTime);
       END_FOR;
       #SyncVal:= PEEK(area := 16#81,
                      dbNumber := 0,
                      byteOffset := 511);
       IF #SyncVal = #CompVal THEN
          GOTO M_1;
       END_IF;
   END_FOR;
   RETURN;

   M_1:
   POKE(area := 16#81,
        dbNumber := 0,
        byteOffset := 511,
        value := B#16#0);
END_FUNCTION

ORGANIZATION_BLOCK "Main"   // OB1, LAD, ProgramCycle
TITLE = "Main Program Sweep (Cycle)"
{ S7_Optimized_Access := 'TRUE' }
VERSION : 0.1
   VAR_INPUT
      Initial_Call : Bool;   // Initial call of this OB
      Remanence : Bool;   // =True, if remanent data are available
   END_VAR
BEGIN

REGION Network 1: FACTORY IO MODULE
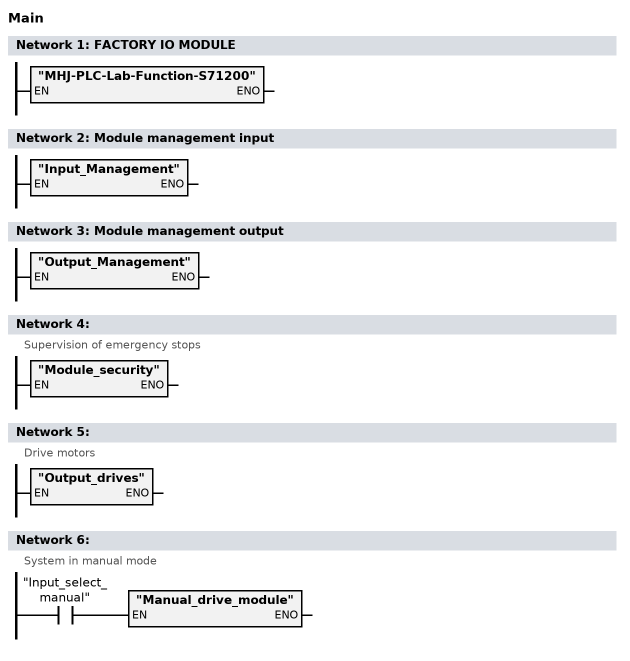
   RUNG wire#powerrail
      "MHJ-PLC-Lab-Function-S71200"()
   END_RUNG
   // the same network as SCL:
   "MHJ-PLC-Lab-Function-S71200"();
END_REGION

REGION Network 2: Module management input
   RUNG wire#powerrail
      "Input_Management"()
   END_RUNG
   // the same network as SCL:
   "Input_Management"();
END_REGION

REGION Network 3: Module management output
   RUNG wire#powerrail
      "Output_Management"()
   END_RUNG
   // the same network as SCL:
   "Output_Management"();
END_REGION

REGION Network 4
   // Supervision of emergency stops
   RUNG wire#powerrail
      "Module_security"()
   END_RUNG
   // the same network as SCL:
   "Module_security"();
END_REGION

REGION Network 5
   // Drive motors
   RUNG wire#powerrail
      "Output_drives"()
   END_RUNG
   // the same network as SCL:
   "Output_drives"();
END_REGION

REGION Network 6
   // System in manual mode
   RUNG wire#powerrail
      Contact( "Input_select_manual" )
      "Manual_drive_module"()
   END_RUNG
   // the same network as SCL:
   IF "Input_select_manual" THEN "Manual_drive_module"(); END_IF;
END_REGION
END_ORGANIZATION_BLOCK